Staubli VAL3: addListItem.pgx

public program addListItem(string& x_sName, string& x_sListName[], string x_sPrefix)
  local string l_sItemName
  local num l_nKey
  local num l_i
  local num l_nPos
begin
  //新建
  do
    call user:listframe("名称",10,5,20,1)
    call user:clear(11,6)
    gotoxy(15,6)
    l_nKey=get(l_sItemName)
    call JudgeSpace(l_i,l_sItemName)
    if l_nKey==270
      //输入为空,赋予一个值
      if l_sItemName==""
        l_i=0
        l_sItemName=x_sPrefix+toString("",l_i+1)
        while l_nPos!=-1
          call FindStr(l_sItemName,x_sListName,l_nPos)
          if l_nPos!=-1
            l_i=l_i+1
            l_sItemName=x_sPrefix+toString("",l_i+1)
          endIf
        endWhile
        x_sName=l_sItemName
      else
        call FindStr(l_sItemName,x_sListName,l_nPos)
        if l_nPos!=-1
          popUpMsg("重复，请重新输入")
          l_sItemName=""
        else
          x_sName=l_sItemName
          return
        endIf
      endIf
    endIf
    delay(0)
  until l_nKey==255
end
